Staubli VAL3: stop.pgx

program stop()
begin
  cls()
  title("End")
  gotoxy(10,7)
  putln(" END Math program")
  resetMotion()
  userPage(false)
end
